PROGRAM MAIN
VAR
//TcRpc tests
	_tcoRtcTest_A						:	TcoRtcTest;
	_tcoRtcTest_B						:	TcoRtcTest;
	_tcoContextTest_A					:	TcoContextTest;
	_tcoContextTest_B					:	TcoContextTest;
	_tcoSequencerAutoRestorableTest		:	TcoSequencerAutoRestorableTest;
	_tcoSequencerNonAutoRestorableTest	:	TcoSequencerNonAutoRestorableTest;
	_tcoMessengerContextTest			:	TcoMessengerContextTest;
	_tcoContextMessagingPerf 			: 	TcoContextMessagingPerf;
	_tcoComponentTest					:	TcoComponentTest;
	_stringBuilderTest					: 	StringBuilderTests;
	
//PLC executed tests
	_tcoTaskTestContext 				:	TcoTaskTestContext;
	_tcoToggleTaskTestContext			:	TcoToggleTaskTestContext;
	{attribute addProperty Name "Test base component class"}
	_tcoComponentTestContext			:   TcoComponentTestContext;
	_tcoRemoteTaskTestContext			:	TcoRemoteTaskTestContext;
	_tcoSequencerTestContext			:	TcoSequencerTestContext;
	_tcoLoggerTestContext				:	TcoLoggerTestContext;
END_VAR

//TcRpc tests
_tcoRtcTest_A();

_tcoRtcTest_B();

_tcoContextTest_A();

_tcoContextTest_B();

_tcoSequencerAutoRestorableTest();

_tcoSequencerNonAutoRestorableTest();

_tcoMessengerContextTest();

_tcoContextMessagingPerf();

_tcoComponentTest();

_stringBuilderTest();

//PLC executed tests
_tcoTaskTestContext.ProbeRun();

_tcoToggleTaskTestContext.ProbeRun();

_tcoComponentTestContext.ProbeRun();

_tcoRemoteTaskTestContext.ProbeRun();

_tcoSequencerTestContext.ProbeRun();

_tcoLoggerTestContext.ProbeRun();

END_PROGRAM

(* stored: Version 1.1.0.1
   POU MAIN: Id {368cd394-e432-4029-bb9d-e4bf92b24162}, SpecialFunc None *)
